// Manages an Event Class, creates an alarm for each Event in the class which can be controlled

// Uses Event Class pre-made in the 'Type System': called 'PersonalEventLogger'
// Uses Events pre-made in the 'Event Class'
// Number of events must be manually defined in '_EventCount'
// Severity of events must be manually defined in '_EventSeverity'

{attribute 'no_explicit_call' := 'Do not call this block directly, use the METHODS this block has'}
FUNCTION_BLOCK EventLogger_Alarms
VAR
	
	_IsRunningToggle		: BOOL;
	_i						: INT;
	
	_Alarm					: ARRAY [1.._EventCount] OF FB_TcAlarm;
	_IsConfirmationNeeded	: ARRAY [1.._EventCount] OF BOOL;
	_Event					: ARRAY [1.._EventCount] OF TcEventEntry;
	_EventSeverity			: ARRAY [1.._EventCount] OF TcEventSeverity := 
								// Manually enter the severity of each alarm here:
								[TcEventSeverity.Error, 
								 TcEventSeverity.Warning];
	
END_VAR
VAR CONSTANT
	
	_EventCount				: INT := 2;

END_VAR

METHOD ClearAlarm : HRESULT
VAR_INPUT
	AlarmId						: UDINT;
	ResetConfirmationState		: BOOL;
END_VAR

// Clears an alarm 

ClearAlarm := _Alarm[AlarmId].Clear(nTimeStamp := 0, bResetConfirmation := ResetConfirmationState);
RETURN;
END_METHOD

METHOD ConfirmAlarm : HRESULT
VAR_INPUT
	AlarmId		: UDINT;
END_VAR

// Acknowledges an alarm 
// This does not clear the alarm
// This does change the alarms state internally

ConfirmAlarm := _Alarm[AlarmId].Confirm(nTimeStamp := 0);
RETURN;
END_METHOD

METHOD CyclicUpdate : BOOL

_IsRunningToggle := NOT(_IsRunningToggle);
RETURN;
END_METHOD

{attribute 'no_explicit_call' := 'You do not need to use this METHOD'}
METHOD FB_init : BOOL 
VAR_INPUT
	bInitRetains : BOOL; // if TRUE, the retain variables are initialized (warm start / cold start)
	bInCopyCode : BOOL;  // if TRUE, the instance afterwards gets moved into the copy code (online change)
END_VAR

// Initialise the event parameters and then the alarms that are tied to the events

FOR _i := 1 TO _EventCount BY 1 DO
	
	// All alarms need confirmation
	_IsConfirmationNeeded[_i] := TRUE;
	
END_FOR

FOR _i := 1 TO _EventCount BY 1 DO
	
	// Defining event settings / parameters
	_Event[_i].uuidEventClass 		:= TC_EVENT_CLASSES.PersonalEventLogger;
	_Event[_i].nEventId 			:= INT_TO_UDINT(_i);
	_Event[_i].eSeverity			:= _EventSeverity[_i];
	
	// Important to set both the Events eFlag and the Alarms bWithConfirmation to the same bool value
	_Event[_i].eFlags 				:= BOOL_TO_BYTE(_IsConfirmationNeeded[_i]);
	
END_FOR

FOR _i := 1 TO _EventCount BY 1 DO

	_Alarm[_i].CreateEx
	(
		stEventEntry := _Event[_i],
		ipSourceInfo := 0,
		
		// Important to set both the Events eFlag and the Alarms bWithConfirmation to the same bool value
		bWithConfirmation := _IsConfirmationNeeded[_i]
	);	

END_FOR

RETURN;
END_METHOD

METHOD Get_AlarmCount : INT // Returns the number of alarms that exist

Get_AlarmCount := _EventCount;
RETURN;
END_METHOD

METHOD Get_AreAlarmsRaised : ARRAY [1.._EventCount] OF BOOL // Returns an array of BOOLS to represent if an alarm is raised

FOR _i := 1 TO _EventCount DO
    Get_AreAlarmsRaised[_i] := _Alarm[_i].bRaised;
END_FOR
RETURN;
END_METHOD

METHOD Get_ConfirmationStates : ARRAY [1.._EventCount] OF TcEventConfirmationState // Returns an array of confirmation states of alarms

FOR _i := 1 TO _EventCount DO
    Get_ConfirmationStates[_i] := _Alarm[_i].eConfirmationState;
END_FOR
RETURN;
END_METHOD

METHOD Get_IsRunningToggle : BOOL // Returns a BOOL that toggles states when the object's cyclic update is running
VAR_INPUT
END_VAR

Get_IsRunningToggle := _IsRunningToggle;
RETURN;
END_METHOD

METHOD TriggerAlarm : HRESULT
VAR_INPUT
	AlarmId		: UDINT;
END_VAR

// Triggers an alarm

TriggerAlarm := _Alarm[AlarmId].Raise(nTimeStamp := 0);
RETURN;
END_METHOD

END_FUNCTION_BLOCK

(* stored: Version 1.1.0.1, ProductVersion 3.1.4024.12
   POU EventLogger_Alarms: Id {adb7947d-436f-4b06-817f-937f8d93f340}, SpecialFunc None
   Method ClearAlarm: Id {17c46d22-1f13-4e66-bbf1-5a792e8c9873}
   Method ConfirmAlarm: Id {7b36f05a-feed-4a82-9307-ccab0ebee3c1}
   Method CyclicUpdate: Id {c4e480e3-9000-4d20-99ed-c0fb37124a08}
   Method FB_init: Id {7c57da50-0899-423f-a02b-0027f2eed138}
   Method Get_AlarmCount: Id {3cb94ad8-0203-4cbf-8705-25f2790828d4}
   Method Get_AreAlarmsRaised: Id {16f8c94b-3c38-41cf-93dc-61541dea3355}
   Method Get_ConfirmationStates: Id {f6e46e15-6287-4803-a798-b1dc11bcf5af}
   Method Get_IsRunningToggle: Id {f07feb80-cf26-431a-b02e-ed5c2448b2de}
   Method TriggerAlarm: Id {f23f0251-0395-401a-8fd8-58d27e94a151} *)
